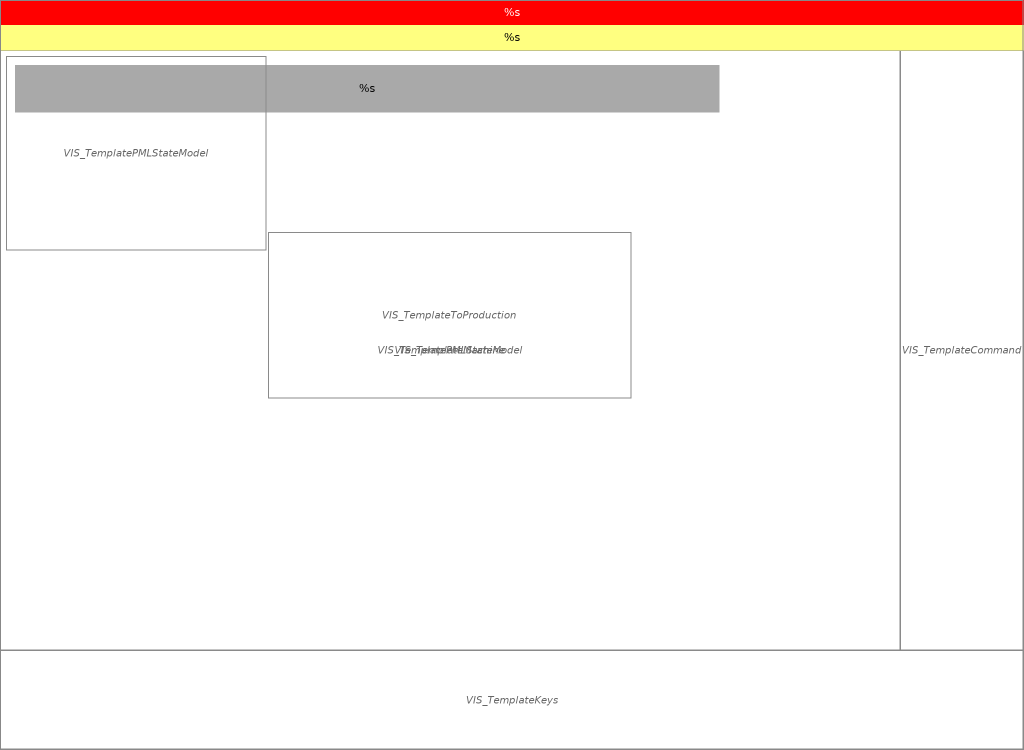
VISUALIZATION visu_main  // 1024x750
    Frame (0,50 900x600), invisible if: MAIN.fbVisu.iFrameVisible = 0 OR MAIN.fbMachine.bChangeIntoProduction
        shows VIS_TemplatePMLStateModel(ePMLUnitMode := MAIN.fbVisu.eModeVisu, ePMLState := MAIN.fbVisu.eStateVisu, eStateCommand := MAIN.fbVisu.eUnitCommand)
        shows VIS_TemplatePMLStateModel()
    Frame (268,232 363x166), invisible if: NOT MAIN.fbMachine.bChangeIntoProduction
        shows VIS_TemplateToProduction(stChangeIntoProduction := GVL.stChangeIntoProduction)
    Textfield (15,65 704x47), "%s", text variable: MAIN.fbVisu.sUnitName, invisible if: MAIN.fbVisu.iFrameVisible = 0 OR MAIN.fbMachine.bChangeIntoProduction
    Frame (0,50 900x600), invisible if: MAIN.fbVisu.iFrameVisible > 0 OR MAIN.fbMachine.bChangeIntoProduction, frame switch variable: G_HMI.iPML_mainFrame
        shows VIS_TemplateMachine()
        shows visu_manual()
    Rectangle (0,0 1024x25), "%s", text variable: MAIN.fbVisu.sAlarmVisu, invisible if: (MAIN.fbMachine.bChangeIntoProduction OR MAIN.fbVisu.sAlarmVisu = '')
    Frame (900,50 124x600)
        shows VIS_TemplateCommand(eModeCommand := GVL.PackTags.Command.UnitMode, eStateCommand := GVL.PackTags.Command.CntrlCmd, eModeStatus := GVL.PackTags.Status.UnitModeCurrent, eStateStatus := GVL.PackTags.Status.StateCurrent, bModeChangeReq := GVL.PackTags.Command.UnitModeChangeRequest)
    Frame (0,650 1024x100)
        shows VIS_TemplateKeys(Caption := GVL.aCaption, KeyPressed := GVL.aKeyPressed)
    Frame (6,56 260x194), invisible if: MAIN.fbVisu.iFrameVisible > 0 OR MAIN.fbMachine.bChangeIntoProduction OR G_HMI.iPML_mainFrame=1
        shows VIS_TemplatePMLStateModel(ePMLUnitMode := GVL.PackTags.Status.UnitModeCurrent, ePMLState := GVL.PackTags.Status.StateCurrent, eStateCommand := MAIN.fbMachine.eCommand)
    Rectangle (0,25 1024x25), "%s", text variable: MAIN.fbVisu.sWarningVisu, invisible if: (MAIN.fbMachine.bChangeIntoProduction OR MAIN.fbVisu.sWarningVisu ='')
END_VISUALIZATION

(* stored: Version 1.1.0.1, ProductVersion 3.1.4024.12
   Visu visu_main: Id {e1801763-8c99-49e1-8dd6-d8ae8e1af5ae} *)
